{attribute 'to_string'}
TYPE e_Device :
(
  General           :=   100,

  CaGroup           :=   200,
  Xpu               :=   300,
  XpuCtrl           :=   400,

  Mover             :=   500,
  MoverCtrl         :=   600,

  XtsTransportUnit  :=   700,

  XtsStation        :=  1000,


  Camming           :=  3000,
  NciChannel        :=  4000,
  NciChannelCtrl    :=  5000,
  Axis              :=  7000,
  Data              := 10000
)DINT;
END_TYPE

(* stored: Version 1.1.0.1, ProductVersion 3.1.4024.12
   DUT e_Device: Id {5ab6f57c-6138-4e8f-b10f-b0f47e40ae34} *)
